Fanuc KAREL source: IO0118.KL

PROGRAM IO0118
%NOLOCKGROUP
ROUTINE RTEST
VAR
  I : INTEGER
  STATUS : INTEGER
  ENTRY : INTEGER
  A : ARRAY[3] OF INTEGER
  B : BOOLEAN
  R : REAL
  P : XYZWPR
  JPOS : JOINTPOS
  PF : POSITION
BEGIN
  I = 1
  A[1] = 2
  B = TRUE
  R = 1.0
  B = RDO[I + 1]
END RTEST
BEGIN
  RTEST
END IO0118
